FUNCTION_BLOCK FB_ElectricityMeter_ABBA44113100
VAR_INPUT
	aElectricityMeterTelegramm	: ARRAY[1..cMBUS_MaxTelegrams] OF ST_MBus_Data2;
END_VAR
VAR_OUTPUT
	fWork : REAL; //Wh
	fPower : REAL; //W
END_VAR
VAR
	{attribute 'OPC.UA.DA' := '1'}
	sensorState : ST_ElectricityMeterState;
END_VAR

sensorState.fWork := STRING_TO_REAL(aElectricityMeterTelegramm[1].arrData[1].sValue);
sensorState.fPower := STRING_TO_REAL(aElectricityMeterTelegramm[2].arrData[1].sValue);

//set outputs
fWork := sensorState.fWork;
fPower := sensorState.fPower;

END_FUNCTION_BLOCK

(* stored: Version 1.1.0.1, ProductVersion 3.1.4024.10
   POU FB_ElectricityMeter_ABBA44113100: Id {a91df6ca-9751-4819-9508-b0844ede8476}, SpecialFunc None *)
